{attribute 'GeneratedUsingTerminal: AMP8000-0030-0103-0103'}
{attribute addProperty BoxType "AMP8000-0030-0103-0103"}
{attribute addProperty Id "FSOEAT %I*FSOE_13BCEA3F2"}
{attribute addProperty CRC "3443497619"}
{attribute addProperty Size "2"}
TYPE FSLOGIC_Inputs_CD3F9A93 :
STRUCT
	{attribute addProperty Name "FSOE"}
	FSOE AT %I* : FSOE_13BCEA3F;
END_STRUCT
END_TYPE

(* stored: Version 1.2.0.0, ProductVersion 3.1.4024.9
   DUT FSLOGIC_Inputs_CD3F9A93: Id {7ded923a-07ce-4b19-9357-41e59965c8e6} *)
